FUNCTION_BLOCK FB_Vector3_Test EXTENDS FB_TestSuite
VAR_INPUT
END_VAR
VAR_OUTPUT
END_VAR
VAR
END_VAR

WhenSetExpectValuesRetained();
WhenReversedExpectValuesReversed();
WhenCrossedExpectVectorOrthogonal();
WhenParallelCrossedExpectCleared();
WhenDottedExpectResult();

METHOD PRIVATE WhenCrossedExpectVectorOrthogonal
VAR_INPUT
END_VAR
VAR
	V1 : Vector3;
	V2 : Vector3;
	V3 : Vector3;
END_VAR
TEST('WhenCrossedExpectVectorOrthogonal');

// @TEST-RUN
V1.SetFromComponents(1,0,0);
V2.SetFromComponents(0,1,0);
V3 := V1.GetVector3CrossProduct(V2);

// @TEST-ASSERT
AssertTrue(V3.Z = 1,'cross product did not work');

TEST_FINISHED();
END_METHOD

METHOD PRIVATE WhenDottedExpectResult
VAR_INPUT
END_VAR
VAR
	V1 : Vector3;
	V2 : Vector3;
	V3 : Vector3;
	Dot : LREAL;
END_VAR
TEST('WhenDottedExpectResult');

// @TEST-RUN
V1.SetFromComponents(1,2,3);
V2 := V1;
Dot := V1.GetVector3DotProduct(V2);

// @TEST-ASSERT
AssertTrue(Dot = 14,'dot product did not work');

TEST_FINISHED();
END_METHOD

METHOD PRIVATE WhenParallelCrossedExpectCleared
VAR_INPUT
END_VAR
VAR
	V1 : Vector3;
	V2 : Vector3;
	V3 : Vector3;
END_VAR
TEST('WhenParallelCrossedExpectCleared');

// @TEST-RUN
V1.SetFromComponents(1,0,0);
V2.SetFromComponents(1,0,0);
V3 := V1.GetVector3CrossProduct(V2);

// @TEST-ASSERT
AssertTrue(V3.IsCleared,'parallel cross product is not zero');

TEST_FINISHED();
END_METHOD

METHOD PRIVATE WhenReversedExpectValuesReversed
VAR_INPUT
END_VAR
VAR
	V1 : Vector3;
	V2 : Vector3;
	V3 : Vector3;
END_VAR
TEST('WhenReversedExpectValuesReversed');

// @TEST-RUN
V1.SetFromComponents(1,2,3);
V2 := V1;
V1 := V1.GetReversed();//tests getter and reverse function
V3 := V2.GetVector3Sum(V2);

// @TEST-ASSERT
AssertTrue(V2.X + V1.X = 0,'Reversal did not work');
AssertTrue(V3.X = 2,'vector sum did not work');

TEST_FINISHED();
END_METHOD

METHOD PRIVATE WhenSetExpectValuesRetained
VAR_INPUT
END_VAR
VAR
	V1 : Vector3;
	V2 : Vector3;
	V3 : DynamicMatrix;
END_VAR
TEST('WhenSetExpectValuesRetained');

// @TEST-RUN
V1.SetFromComponents(1,2,3);
V2 := V1;
V1.Clear();
V3.InitVector(3,1,1);

// @TEST-ASSERT
AssertTrue(V2.z = 3,'Component access not retained');
AssertTrue(V2.IsEqual(V3),'vector did not copy');

TEST_FINISHED();
END_METHOD

END_FUNCTION_BLOCK

(* stored: Version 1.1.0.1, ProductVersion 3.1.4024.9
   POU FB_Vector3_Test: Id {13478125-18c9-4a6b-bc64-7376bfcd3840}, SpecialFunc None
   Method WhenCrossedExpectVectorOrthogonal: Id {77217c58-9dca-41bd-bf6e-dd652b36e1c1}
   Method WhenDottedExpectResult: Id {9668ad9e-694a-4131-b760-7aa5f1e21bae}
   Method WhenParallelCrossedExpectCleared: Id {26b6e7b2-0fd1-05df-0e33-19e6d7a942cd}
   Method WhenReversedExpectValuesReversed: Id {3f55f92d-d03c-47e6-ab90-b6404c9d174c}
   Method WhenSetExpectValuesRetained: Id {bc97fc39-a708-467e-8709-58aa23a1fcd5} *)
